ADAPTER ModbusBusAdapter (* Modbus Bus Adapter *)
  (* Standard: 61499-1; Description: Copyright (c) 2024 Martin Erich Jobst This program and the accompanying materials are made available under the terms of the Eclipse Public License 2.0 which is available at https://www.eclipse.org/legal/epl-2.0/ SPDX-License-Identifier: EPL-2.0 *)
  (* Version 1.0, 2024-09-12, Martin Erich Jobst *)
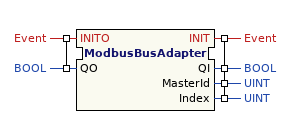
  EVENT_INPUT
    INITO WITH QO;
  END_EVENT
  EVENT_OUTPUT
    INIT WITH QI, MasterId, Index;
  END_EVENT
  VAR_INPUT
    QO : BOOL;
  END_VAR
  VAR_OUTPUT
    QI : BOOL;
    MasterId : UINT;
    Index : UINT;
  END_VAR
END_ADAPTER
